// Mitsubishi GX Works2 project: Lamp_control_2   PLC: Q03UDV

PROGRAM MAIN
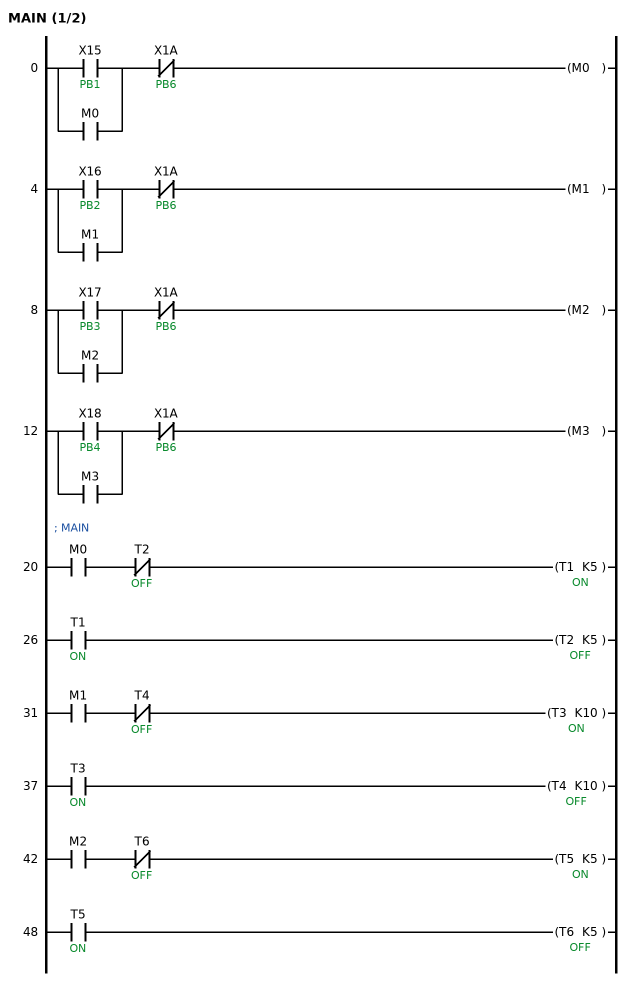
0     LD      X15  ; PB1
      OR      M0
      ANI     X1A  ; PB6
      OUT     M0
4     LD      X16  ; PB2
      OR      M1
      ANI     X1A  ; PB6
      OUT     M1
8     LD      X17  ; PB3
      OR      M2
      ANI     X1A  ; PB6
      OUT     M2
12    LD      X18  ; PB4
      OR      M3
      ANI     X1A  ; PB6
      OUT     M3
; MAIN
20    LD      M0
      ANI     T2  ; OFF
      OUT     T1 K5  ; ON
26    LD      T1  ; ON
      OUT     T2 K5  ; OFF
31    LD      M1
      ANI     T4  ; OFF
      OUT     T3 K10  ; ON
37    LD      T3  ; ON
      OUT     T4 K10  ; OFF
42    LD      M2
      ANI     T6  ; OFF
      OUT     T5 K5  ; ON
48    LD      T5  ; ON
      OUT     T6 K5  ; OFF
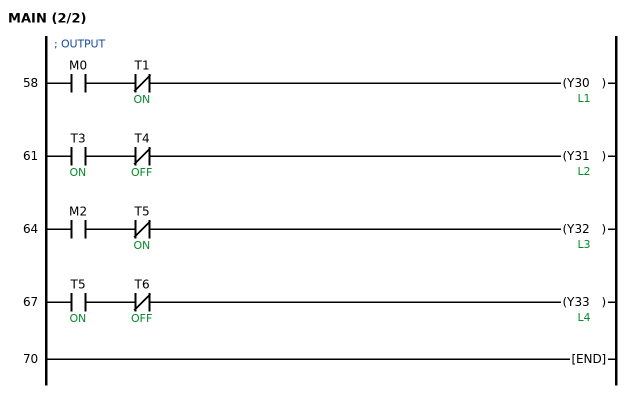
; OUTPUT
58    LD      M0
      ANI     T1  ; ON
      OUT     Y30  ; L1
61    LD      T3  ; ON
      ANI     T4  ; OFF
      OUT     Y31  ; L2
64    LD      M2
      ANI     T5  ; ON
      OUT     Y32  ; L3
67    LD      T5  ; ON
      ANI     T6  ; OFF
      OUT     Y33  ; L4
70    END
END_PROGRAM

// device comments not shown above
X1  ; RS1-1
X2  ; RS1-2
X3  ; RS2-1
X4  ; RS2-2
X19  ; PB5
X1B  ; PB7
X1C  ; X1B
Y34  ; L5
Y35  ; L6
Y36  ; L7
Y37  ; BUZZER
Y38  ; S/V1-1
Y39  ; S/V1-2
Y3A  ; S/V2
M10  ; KILL
T7  ; A
T8  ; B
T9  ; C
